LIN {X 0,Y 156.4,Z 371.31,A -85,B 0,C 180,E1 -29332.253,E2 -29332.253} C_VEL
LIN {X 0,Y 156.384,Z 371.279,A -85,B 0,C 180,E1 -29334.844,E2 -29334.844} C_VEL
LIN {X 0,Y 156.569,Z 371.648,A -85,B 0,C 180,E1 -29337.428,E2 -29337.428} C_VEL
LIN {X 0,Y 156.555,Z 373.641,A -85,B 0,C 180,E1 -29340.209,E2 -29340.209} C_VEL
LIN {X 0,Y 155.258,Z 377.324,A -85,B 0,C 180,E1 -29340.488,E2 -29340.488} C_VEL
LIN {X 0,Y 149.876,Z 389.562,A -85,B 0,C 180,E1 -29341.234,E2 -29341.234} C_VEL
LIN {X 0,Y 144.167,Z 399.757,A -85,B 0,C 180,E1 -29342.148,E2 -29342.148} C_VEL
LIN {X 0,Y 137.568,Z 409.301,A -85,B 0,C 180,E1 -29343.179,E2 -29343.179} C_VEL
LIN {X 0,Y 133.867,Z 413.861,A -85,B 0,C 180,E1 -29343.493,E2 -29343.493} C_VEL
LIN {X 0,Y 126.954,Z 420.984,A -85,B 0,C 180,E1 -29343.346,E2 -29343.346} C_VEL
LIN {X 0,Y 119.532,Z 427.573,A -85,B 0,C 180,E1 -29343.286,E2 -29343.286} C_VEL
LIN {X 0,Y 115.039,Z 431.197,A -85,B 0,C 180,E1 -29343.819,E2 -29343.819} C_VEL
LIN {X 0,Y 105.964,Z 437.725,A -85,B 0,C 180,E1 -29345.853,E2 -29345.853} C_VEL
LIN {X 0,Y 96.194,Z 443.469,A -85,B 0,C 180,E1 -29348.403,E2 -29348.403} C_VEL
LIN {X 0,Y 86.151,Z 448.159,A -85,B 0,C 180,E1 -29351.809,E2 -29351.809} C_VEL
LIN {X 0,Y 76.542,Z 451.58,A -85,B 0,C 180,E1 -29355.991,E2 -29355.991} C_VEL
LIN {X 0,Y 67.777,Z 453.839,A -85,B 0,C 180,E1 -29361.075,E2 -29361.075} C_VEL
LIN {X 0,Y 58.641,Z 455.229,A -85,B 0,C 180,E1 -29368.648,E2 -29368.648} C_VEL
LIN {X 0,Y 52.297,Z 455.5,A -85,B 0,C 180,E1 -29376.277,E2 -29376.277} C_VEL
LIN {X 0,Y 45.048,Z 454.461,A -85,B 0,C 180,E1 -29391.27,E2 -29391.27} C_VEL
LIN {X 0,Y 42.636,Z 453.317,A -85,B 0,C 180,E1 -29400.374,E2 -29400.374} C_VEL
LIN {X 0,Y 41.077,Z 450.774,A -85,B 0,C 180,E1 -29415.141,E2 -29415.141} C_VEL
LIN {X 0,Y 42.17,Z 447.189,A -85,B 0,C 180,E1 -29430.011,E2 -29430.011} C_VEL
LIN {X 0,Y 45.323,Z 442.498,A -85,B 0,C 180,E1 -29443.46,E2 -29443.46} C_VEL
LIN {X 0,Y 50.177,Z 436.573,A -85,B 0,C 180,E1 -29454.856,E2 -29454.856} C_VEL
LIN {X 0,Y 56.499,Z 429.187,A -85,B 0,C 180,E1 -29464.049,E2 -29464.049} C_VEL
LIN {X 0,Y 62.629,Z 421.633,A -85,B 0,C 180,E1 -29470.193,E2 -29470.193} C_VEL
LIN {X 0,Y 69.244,Z 412.469,A -85,B 0,C 180,E1 -29475.282,E2 -29475.282} C_VEL
LIN {X 0,Y 75.578,Z 402.269,A -85,B 0,C 180,E1 -29479.081,E2 -29479.081} C_VEL
LIN {X 0,Y 81.46,Z 390.96,A -85,B 0,C 180,E1 -29481.939,E2 -29481.939} C_VEL
LIN {X 0,Y 85.753,Z 380.375,A -85,B 0,C 180,E1 -29483.986,E2 -29483.986} C_VEL
LIN {X 0,Y 88.852,Z 370.817,A -85,B 0,C 180,E1 -29485.293,E2 -29485.293} C_VEL
LIN {X 0,Y 88.467,Z 370.007,A -85,B 0,C 180,E1 -29486.212,E2 -29486.212} C_VEL
LIN {X 0,Y 84.653,Z 375.313,A -85,B 0,C 180,E1 -29488.741,E2 -29488.741} C_VEL
LIN {X 0,Y 82.326,Z 378.124,A -85,B 0,C 180,E1 -29490.602,E2 -29490.602} C_VEL
LIN {X 0,Y 77.718,Z 385.279,A -85,B 0,C 180,E1 -29493.117,E2 -29493.117} C_VEL
LIN {X 0,Y 73.643,Z 390.721,A -85,B 0,C 180,E1 -29496.07,E2 -29496.07} C_VEL
LIN {X 0,Y 69.306,Z 395.953,A -85,B 0,C 180,E1 -29500.486,E2 -29500.486} C_VEL
LIN {X 0,Y 66.79,Z 398.707,A -85,B 0,C 180,E1 -29504.746,E2 -29504.746} C_VEL
LIN {X 0,Y 65.658,Z 400.025,A -85,B 0,C 180,E1 -29507.637,E2 -29507.637} C_VEL
LIN {X 0,Y 61.447,Z 406.178,A -85,B 0,C 180,E1 -29515.077,E2 -29515.077} C_VEL
LIN {X 0,Y 59.957,Z 408.868,A -85,B 0,C 180,E1 -29519.998,E2 -29519.998} C_VEL
LIN {X 0,Y 59.696,Z 412.054,A -85,B 0,C 180,E1 -29529.306,E2 -29529.306} C_VEL
LIN {X 0,Y 58.943,Z 418.506,A -85,B 0,C 180,E1 -29540.958,E2 -29540.958} C_VEL
LIN {X 0,Y 61.299,Z 422.846,A -85,B 0,C 180,E1 -29551.058,E2 -29551.058} C_VEL
LIN {X 0,Y 66.387,Z 425.676,A -85,B 0,C 180,E1 -29559.432,E2 -29559.432} C_VEL
LIN {X 0,Y 65.129,Z 427.629,A -85,B 0,C 180,E1 -29560.932,E2 -29560.932} C_VEL
LIN {X 0,Y 58.025,Z 434.595,A -85,B 0,C 180,E1 -29565.847,E2 -29565.847} C_VEL
LIN {X 0,Y 50.876,Z 441.526,A -85,B 0,C 180,E1 -29574.039,E2 -29574.039} C_VEL
LIN {X 0,Y 46.337,Z 446.235,A -85,B 0,C 180,E1 -29582.924,E2 -29582.924} C_VEL
LIN {X 0,Y 42.935,Z 450.806,A -85,B 0,C 180,E1 -29595.776,E2 -29595.776} C_VEL
LIN {X 0,Y 41.947,Z 454.261,A -85,B 0,C 180,E1 -29609.989,E2 -29609.989} C_VEL
LIN {X 0,Y 41.814,Z 455.932,A -85,B 0,C 180,E1 -29619.665,E2 -29619.665} C_VEL
LIN {X 0,Y 44.823,Z 458.027,A -85,B 0,C 180,E1 -29638.048,E2 -29638.048} C_VEL
LIN {X 0,Y 47.781,Z 458.503,A -85,B 0,C 180,E1 -29646.029,E2 -29646.029} C_VEL
LIN {X 0,Y 56.157,Z 458.254,A -85,B 0,C 180,E1 -29658.655,E2 -29658.655} C_VEL
LIN {X 0,Y 66.548,Z 456.484,A -85,B 0,C 180,E1 -29667.644,E2 -29667.644} C_VEL
LIN {X 0,Y 72.208,Z 454.987,A -85,B 0,C 180,E1 -29671.146,E2 -29671.146} C_VEL
LIN {X 0,Y 81.173,Z 451.969,A -85,B 0,C 180,E1 -29675.367,E2 -29675.367} C_VEL
LIN {X 0,Y 90.543,Z 447.926,A -85,B 0,C 180,E1 -29678.648,E2 -29678.648} C_VEL
LIN {X 0,Y 101.823,Z 441.734,A -85,B 0,C 180,E1 -29681.617,E2 -29681.617} C_VEL
LIN {X 0,Y 111.69,Z 435.017,A -85,B 0,C 180,E1 -29683.641,E2 -29683.641} C_VEL
LIN {X 0,Y 120.018,Z 428.188,A -85,B 0,C 180,E1 -29685.047,E2 -29685.047} C_VEL
LIN {X 0,Y 128.391,Z 419.99,A -85,B 0,C 180,E1 -29686.301,E2 -29686.301} C_VEL
LIN {X 0,Y 136.884,Z 409.9,A -85,B 0,C 180,E1 -29687.278,E2 -29687.278} C_VEL
LIN {X 0,Y 144.569,Z 398.566,A -85,B 0,C 180,E1 -29688.015,E2 -29688.015} C_VEL
LIN {X 0,Y 150.579,Z 387.394,A -85,B 0,C 180,E1 -29688.544,E2 -29688.544} C_VEL
LIN {X 0,Y 153.767,Z 379.997,A -85,B 0,C 180,E1 -29688.827,E2 -29688.827} C_VEL
LIN {X 0,Y 154.098,Z 378.981,A -85,B 0,C 180,E1 -29689.157,E2 -29689.157} C_VEL
LIN {X 0,Y 154.001,Z 378.017,A -85,B 0,C 180,E1 -29692.132,E2 -29692.132} C_VEL
LIN {X 0,Y 153.959,Z 377.955,A -85,B 0,C 180,E1 -29694.762,E2 -29694.762} C_VEL
LIN {X 0,Y 154,Z 378.711,A -85,B 0,C 180,E1 -29697.73,E2 -29697.73} C_VEL
LIN {X 0,Y 152.902,Z 381.549,A -85,B 0,C 180,E1 -29698.062,E2 -29698.062} C_VEL
LIN {X 0,Y 147.616,Z 392.5,A -85,B 0,C 180,E1 -29698.73,E2 -29698.73} C_VEL
LIN {X 0,Y 140.553,Z 404.019,A -85,B 0,C 180,E1 -29699.702,E2 -29699.702} C_VEL
LIN {X 0,Y 132.658,Z 414.293,A -85,B 0,C 180,E1 -29700.794,E2 -29700.794} C_VEL
LIN {X 0,Y 123.085,Z 424.288,A -85,B 0,C 180,E1 -29702.343,E2 -29702.343} C_VEL
LIN {X 0,Y 115.039,Z 431.197,A -85,B 0,C 180,E1 -29703.819,E2 -29703.819} C_VEL
LIN {X 0,Y 110.384,Z 434.655,A -85,B 0,C 180,E1 -29704.426,E2 -29704.426} C_VEL
LIN {X 0,Y 101.975,Z 439.939,A -85,B 0,C 180,E1 -29704.627,E2 -29704.627} C_VEL
LIN {X 0,Y 93.209,Z 444.505,A -85,B 0,C 180,E1 -29704.971,E2 -29704.971} C_VEL
LIN {X 0,Y 88.028,Z 446.834,A -85,B 0,C 180,E1 -29705.963,E2 -29705.963} C_VEL
LIN {X 0,Y 78.299,Z 450.562,A -85,B 0,C 180,E1 -29709.164,E2 -29709.164} C_VEL
LIN {X 0,Y 71.797,Z 452.509,A -85,B 0,C 180,E1 -29711.83,E2 -29711.83} C_VEL
LIN {X 0,Y 65.475,Z 454.015,A -85,B 0,C 180,E1 -29715.001,E2 -29715.001} C_VEL
LIN {X 0,Y 54.483,Z 455.57,A -85,B 0,C 180,E1 -29722.769,E2 -29722.769} C_VEL
LIN {X 0,Y 48.298,Z 455.832,A -85,B 0,C 180,E1 -29729.2,E2 -29729.2} C_VEL
LIN {X 0,Y 43.512,Z 455.567,A -85,B 0,C 180,E1 -29736.156,E2 -29736.156} C_VEL
LIN {X 0,Y 38.983,Z 454.745,A -85,B 0,C 180,E1 -29746.152,E2 -29746.152} C_VEL
LIN {X 0,Y 34.502,Z 452.265,A -85,B 0,C 180,E1 -29765.973,E2 -29765.973} C_VEL
LIN {X 0,Y 34.273,Z 449.12,A -85,B 0,C 180,E1 -29784.128,E2 -29784.128} C_VEL
LIN {X 0,Y 36.969,Z 444.898,A -85,B 0,C 180,E1 -29800.971,E2 -29800.971} C_VEL
LIN {X 0,Y 41.814,Z 439.512,A -85,B 0,C 180,E1 -29814.858,E2 -29814.858} C_VEL
LIN {X 0,Y 48.329,Z 432.775,A -85,B 0,C 180,E1 -29825.579,E2 -29825.579} C_VEL
LIN {X 0,Y 55.995,Z 424.373,A -85,B 0,C 180,E1 -29833.665,E2 -29833.665} C_VEL
LIN {X 0,Y 63,Z 415.704,A -85,B 0,C 180,E1 -29838.861,E2 -29838.861} C_VEL
LIN {X 0,Y 70.402,Z 405.048,A -85,B 0,C 180,E1 -29843.009,E2 -29843.009} C_VEL
LIN {X 0,Y 76.535,Z 394.349,A -85,B 0,C 180,E1 -29845.745,E2 -29845.745} C_VEL
LIN {X 0,Y 79.81,Z 387.444,A -85,B 0,C 180,E1 -29847.116,E2 -29847.116} C_VEL
LIN {X 0,Y 79.516,Z 387.02,A -85,B 0,C 180,E1 -29847.972,E2 -29847.972} C_VEL
LIN {X 0,Y 74.252,Z 393.462,A -85,B 0,C 180,E1 -29850.764,E2 -29850.764} C_VEL
LIN {X 0,Y 69.473,Z 398.568,A -85,B 0,C 180,E1 -29854.317,E2 -29854.317} C_VEL
LIN {X 0,Y 65.913,Z 402.042,A -85,B 0,C 180,E1 -29858.086,E2 -29858.086} C_VEL
LIN {X 0,Y 62.721,Z 404.943,A -85,B 0,C 180,E1 -29863.731,E2 -29863.731} C_VEL
LIN {X 0,Y 58.027,Z 410.485,A -85,B 0,C 180,E1 -29870.805,E2 -29870.805} C_VEL
LIN {X 0,Y 55.959,Z 413.213,A -85,B 0,C 180,E1 -29876.037,E2 -29876.037} C_VEL
LIN {X 0,Y 54.662,Z 416.981,A -85,B 0,C 180,E1 -29887.385,E2 -29887.385} C_VEL
LIN {X 0,Y 53.417,Z 422.478,A -85,B 0,C 180,E1 -29898.885,E2 -29898.885} C_VEL
LIN {X 0,Y 55.357,Z 426.811,A -85,B 0,C 180,E1 -29910.518,E2 -29910.518} C_VEL
LIN {X 0,Y 58.393,Z 428.778,A -85,B 0,C 180,E1 -29916.996,E2 -29916.996} C_VEL
LIN {X 0,Y 50.417,Z 436.169,A -85,B 0,C 180,E1 -29922.946,E2 -29922.946} C_VEL
LIN {X 0,Y 44.233,Z 441.735,A -85,B 0,C 180,E1 -29930.527,E2 -29930.527} C_VEL
LIN {X 0,Y 38.535,Z 447.18,A -85,B 0,C 180,E1 -29942.861,E2 -29942.861} C_VEL
LIN {X 0,Y 35.368,Z 451.453,A -85,B 0,C 180,E1 -29958.526,E2 -29958.526} C_VEL
LIN {X 0,Y 34.861,Z 453.696,A -85,B 0,C 180,E1 -29969.987,E2 -29969.987} C_VEL
LIN {X 0,Y 34.827,Z 455.438,A -85,B 0,C 180,E1 -29981.629,E2 -29981.629} C_VEL
LIN {X 0,Y 38.665,Z 457.615,A -85,B 0,C 180,E1 -30003.032,E2 -30003.032} C_VEL
LIN {X 0,Y 46.691,Z 458.274,A -85,B 0,C 180,E1 -30018.801,E2 -30018.801} C_VEL
LIN {X 0,Y 57.221,Z 457.338,A -85,B 0,C 180,E1 -30029.273,E2 -30029.273} C_VEL
LIN {X 0,Y 69.052,Z 454.878,A -85,B 0,C 180,E1 -30036.332,E2 -30036.332} C_VEL
LIN {X 0,Y 78.478,Z 451.931,A -85,B 0,C 180,E1 -30040.087,E2 -30040.087} C_VEL
LIN {X 0,Y 88.204,Z 447.974,A -85,B 0,C 180,E1 -30042.95,E2 -30042.95} C_VEL
LIN {X 0,Y 98.142,Z 442.893,A -85,B 0,C 180,E1 -30045.163,E2 -30045.163} C_VEL
LIN {X 0,Y 108.2,Z 436.508,A -85,B 0,C 180,E1 -30046.964,E2 -30046.964} C_VEL
LIN {X 0,Y 118.391,Z 428.578,A -85,B 0,C 180,E1 -30048.354,E2 -30048.354} C_VEL
LIN {X 0,Y 126.905,Z 420.521,A -85,B 0,C 180,E1 -30049.399,E2 -30049.399} C_VEL
LIN {X 0,Y 135.504,Z 410.688,A -85,B 0,C 180,E1 -30050.193,E2 -30050.193} C_VEL
LIN {X 0,Y 143.159,Z 399.774,A -85,B 0,C 180,E1 -30050.772,E2 -30050.772} C_VEL
LIN {X 0,Y 149.87,Z 387.705,A -85,B 0,C 180,E1 -30051.236,E2 -30051.236} C_VEL
LIN {X 0,Y 150.401,Z 386.6,A -85,B 0,C 180,E1 -30051.275,E2 -30051.275} C_VEL
LIN {X 0,Y 151.219,Z 384.614,A -85,B 0,C 180,E1 -30051.986,E2 -30051.986} C_VEL
LIN {X 0,Y 151.157,Z 384.597,A -85,B 0,C 180,E1 -30055.312,E2 -30055.312} C_VEL
LIN {X 0,Y 150.66,Z 385.733,A -85,B 0,C 180,E1 -30055.592,E2 -30055.592} C_VEL
LIN {X 0,Y 144.371,Z 397.448,A -85,B 0,C 180,E1 -30056.274,E2 -30056.274} C_VEL
LIN {X 0,Y 137.393,Z 407.735,A -85,B 0,C 180,E1 -30057.069,E2 -30057.069} C_VEL
LIN {X 0,Y 130.093,Z 416.564,A -85,B 0,C 180,E1 -30057.945,E2 -30057.945} C_VEL
LIN {X 0,Y 121.238,Z 425.413,A -85,B 0,C 180,E1 -30059.163,E2 -30059.163} C_VEL
LIN {X 0,Y 110.695,Z 433.897,A -85,B 0,C 180,E1 -30060.839,E2 -30060.839} C_VEL
LIN {X 0,Y 100.268,Z 440.649,A -85,B 0,C 180,E1 -30062.887,E2 -30062.887} C_VEL
LIN {X 0,Y 91.696,Z 445.155,A -85,B 0,C 180,E1 -30064.939,E2 -30064.939} C_VEL
LIN {X 0,Y 88.028,Z 446.834,A -85,B 0,C 180,E1 -30065.963,E2 -30065.963} C_VEL
LIN {X 0,Y 82.761,Z 448.953,A -85,B 0,C 180,E1 -30067.113,E2 -30067.113} C_VEL
LIN {X 0,Y 73.38,Z 451.955,A -85,B 0,C 180,E1 -30068.05,E2 -30068.05} C_VEL
LIN {X 0,Y 63.849,Z 454.195,A -85,B 0,C 180,E1 -30069.298,E2 -30069.298} C_VEL
LIN {X 0,Y 58.437,Z 455.085,A -85,B 0,C 180,E1 -30071.281,E2 -30071.281} C_VEL
LIN {X 0,Y 50.936,Z 455.914,A -85,B 0,C 180,E1 -30076.021,E2 -30076.021} C_VEL
LIN {X 0,Y 45.151,Z 456.14,A -85,B 0,C 180,E1 -30080.971,E2 -30080.971} C_VEL
LIN {X 0,Y 39.6,Z 455.956,A -85,B 0,C 180,E1 -30087.479,E2 -30087.479} C_VEL
LIN {X 0,Y 33.326,Z 455.026,A -85,B 0,C 180,E1 -30099.25,E2 -30099.25} C_VEL
LIN {X 0,Y 27.969,Z 452.815,A -85,B 0,C 180,E1 -30119.85,E2 -30119.85} C_VEL
LIN {X 0,Y 27.023,Z 449.758,A -85,B 0,C 180,E1 -30142.545,E2 -30142.545} C_VEL
LIN {X 0,Y 29.943,Z 445.621,A -85,B 0,C 180,E1 -30163.59,E2 -30163.59} C_VEL
LIN {X 0,Y 36.554,Z 439.323,A -85,B 0,C 180,E1 -30181.933,E2 -30181.933} C_VEL
LIN {X 0,Y 44.061,Z 432.474,A -85,B 0,C 180,E1 -30192.693,E2 -30192.693} C_VEL
LIN {X 0,Y 51.075,Z 425.472,A -85,B 0,C 180,E1 -30199.197,E2 -30199.197} C_VEL
LIN {X 0,Y 58.577,Z 416.977,A -85,B 0,C 180,E1 -30204.094,E2 -30204.094} C_VEL
LIN {X 0,Y 65.275,Z 408.121,A -85,B 0,C 180,E1 -30207.427,E2 -30207.427} C_VEL
LIN {X 0,Y 68.189,Z 403.722,A -85,B 0,C 180,E1 -30208.742,E2 -30208.742} C_VEL
LIN {X 0,Y 68.918,Z 402.36,A -85,B 0,C 180,E1 -30209.342,E2 -30209.342} C_VEL
LIN {X 0,Y 63.714,Z 406.759,A -85,B 0,C 180,E1 -30213.816,E2 -30213.816} C_VEL
LIN {X 0,Y 59.897,Z 409.646,A -85,B 0,C 180,E1 -30219.388,E2 -30219.388} C_VEL
LIN {X 0,Y 55.228,Z 414.152,A -85,B 0,C 180,E1 -30225.254,E2 -30225.254} C_VEL
LIN {X 0,Y 51.801,Z 417.679,A -85,B 0,C 180,E1 -30232.2,E2 -30232.2} C_VEL
LIN {X 0,Y 49.42,Z 421.752,A -85,B 0,C 180,E1 -30245.366,E2 -30245.366} C_VEL
LIN {X 0,Y 47.797,Z 426.491,A -85,B 0,C 180,E1 -30257.1,E2 -30257.1} C_VEL
LIN {X 0,Y 49.29,Z 430.523,A -85,B 0,C 180,E1 -30269.94,E2 -30269.94} C_VEL
LIN {X 0,Y 50.186,Z 431.333,A -85,B 0,C 180,E1 -30272.82,E2 -30272.82} C_VEL
LIN {X 0,Y 48.924,Z 432.719,A -85,B 0,C 180,E1 -30274.294,E2 -30274.294} C_VEL
LIN {X 0,Y 40.327,Z 439.869,A -85,B 0,C 180,E1 -30282.196,E2 -30282.196} C_VEL
LIN {X 0,Y 32.395,Z 446.487,A -85,B 0,C 180,E1 -30297.139,E2 -30297.139} C_VEL
LIN {X 0,Y 28.459,Z 450.847,A -85,B 0,C 180,E1 -30315.687,E2 -30315.687} C_VEL
LIN {X 0,Y 27.76,Z 453.131,A -85,B 0,C 180,E1 -30329.984,E2 -30329.984} C_VEL
LIN {X 0,Y 27.893,Z 454.917,A -85,B 0,C 180,E1 -30344.577,E2 -30344.577} C_VEL
LIN {X 0,Y 29.713,Z 456.275,A -85,B 0,C 180,E1 -30358.216,E2 -30358.216} C_VEL
LIN {X 0,Y 37.205,Z 457.757,A -85,B 0,C 180,E1 -30379.059,E2 -30379.059} C_VEL
LIN {X 0,Y 47.943,Z 457.737,A -85,B 0,C 180,E1 -30391.568,E2 -30391.568} C_VEL
LIN {X 0,Y 60.136,Z 456.121,A -85,B 0,C 180,E1 -30399.199,E2 -30399.199} C_VEL
LIN {X 0,Y 66.51,Z 454.742,A -85,B 0,C 180,E1 -30401.969,E2 -30401.969} C_VEL
LIN {X 0,Y 76.348,Z 451.871,A -85,B 0,C 180,E1 -30405.114,E2 -30405.114} C_VEL
LIN {X 0,Y 86.39,Z 447.999,A -85,B 0,C 180,E1 -30407.455,E2 -30407.455} C_VEL
LIN {X 0,Y 96.57,Z 443.016,A -85,B 0,C 180,E1 -30409.232,E2 -30409.232} C_VEL
LIN {X 0,Y 106.824,Z 436.772,A -85,B 0,C 180,E1 -30410.673,E2 -30410.673} C_VEL
LIN {X 0,Y 117.17,Z 428.969,A -85,B 0,C 180,E1 -30411.738,E2 -30411.738} C_VEL
LIN {X 0,Y 125.797,Z 421.052,A -85,B 0,C 180,E1 -30412.562,E2 -30412.562} C_VEL
LIN {X 0,Y 134.481,Z 411.397,A -85,B 0,C 180,E1 -30413.16,E2 -30413.16} C_VEL
LIN {X 0,Y 141.451,Z 401.94,A -85,B 0,C 180,E1 -30413.537,E2 -30413.537} C_VEL
LIN {X 0,Y 141.399,Z 401.999,A -85,B 0,C 180,E1 -30413.723,E2 -30413.723} C_VEL
LIN {X 0,Y 133.27,Z 412.765,A -85,B 0,C 180,E1 -30414.45,E2 -30414.45} C_VEL
LIN {X 0,Y 125.161,Z 421.52,A -85,B 0,C 180,E1 -30415.293,E2 -30415.293} C_VEL
LIN {X 0,Y 116.801,Z 429,A -85,B 0,C 180,E1 -30416.244,E2 -30416.244} C_VEL
LIN {X 0,Y 107.267,Z 436.069,A -85,B 0,C 180,E1 -30417.542,E2 -30417.542} C_VEL
LIN {X 0,Y 98.399,Z 441.468,A -85,B 0,C 180,E1 -30418.977,E2 -30418.977} C_VEL
LIN {X 0,Y 87.857,Z 446.669,A -85,B 0,C 180,E1 -30421.075,E2 -30421.075} C_VEL
LIN {X 0,Y 77.465,Z 450.611,A -85,B 0,C 180,E1 -30423.743,E2 -30423.743} C_VEL
LIN {X 0,Y 70.652,Z 452.603,A -85,B 0,C 180,E1 -30425.949,E2 -30425.949} C_VEL
LIN {X 0,Y 63.958,Z 454.161,A -85,B 0,C 180,E1 -30428.571,E2 -30428.571} C_VEL
LIN {X 0,Y 58.437,Z 455.085,A -85,B 0,C 180,E1 -30431.281,E2 -30431.281} C_VEL
LIN {X 0,Y 53.057,Z 455.8,A -85,B 0,C 180,E1 -30433.681,E2 -30433.681} C_VEL
LIN {X 0,Y 43.505,Z 456.321,A -85,B 0,C 180,E1 -30436.814,E2 -30436.814} C_VEL
LIN {X 0,Y 34.122,Z 456.06,A -85,B 0,C 180,E1 -30441.645,E2 -30441.645} C_VEL
LIN {X 0,Y 29.3,Z 455.471,A -85,B 0,C 180,E1 -30447.775,E2 -30447.775} C_VEL
LIN {X 0,Y 21.953,Z 453.335,A -85,B 0,C 180,E1 -30470.215,E2 -30470.215} C_VEL
LIN {X 0,Y 19.819,Z 450.365,A -85,B 0,C 180,E1 -30499.81,E2 -30499.81} C_VEL
LIN {X 0,Y 22.982,Z 446.33,A -85,B 0,C 180,E1 -30527.827,E2 -30527.827} C_VEL
LIN {X 0,Y 30.726,Z 440.141,A -85,B 0,C 180,E1 -30548.996,E2 -30548.996} C_VEL
LIN {X 0,Y 39.11,Z 433.403,A -85,B 0,C 180,E1 -30559.811,E2 -30559.811} C_VEL
LIN {X 0,Y 48.304,Z 424.999,A -85,B 0,C 180,E1 -30566.799,E2 -30566.799} C_VEL
LIN {X 0,Y 56.314,Z 416.328,A -85,B 0,C 180,E1 -30570.896,E2 -30570.896} C_VEL
LIN {X 0,Y 57.932,Z 414.399,A -85,B 0,C 180,E1 -30571.602,E2 -30571.602} C_VEL
LIN {X 0,Y 57.483,Z 413.986,A -85,B 0,C 180,E1 -30574.216,E2 -30574.216} C_VEL
LIN {X 0,Y 49.692,Z 420.22,A -85,B 0,C 180,E1 -30583.567,E2 -30583.567} C_VEL
LIN {X 0,Y 46.478,Z 423.056,A -85,B 0,C 180,E1 -30591.301,E2 -30591.301} C_VEL
LIN {X 0,Y 44.594,Z 425.344,A -85,B 0,C 180,E1 -30599.998,E2 -30599.998} C_VEL
LIN {X 0,Y 42.692,Z 428.404,A -85,B 0,C 180,E1 -30608.925,E2 -30608.925} C_VEL
LIN {X 0,Y 42.279,Z 432.649,A -85,B 0,C 180,E1 -30623.891,E2 -30623.891} C_VEL
LIN {X 0,Y 42.309,Z 434.236,A -85,B 0,C 180,E1 -30628.689,E2 -30628.689} C_VEL
LIN {X 0,Y 33.12,Z 441.153,A -85,B 0,C 180,E1 -30637.252,E2 -30637.252} C_VEL
LIN {X 0,Y 24.671,Z 447.382,A -85,B 0,C 180,E1 -30655.247,E2 -30655.247} C_VEL
LIN {X 0,Y 20.939,Z 451.46,A -85,B 0,C 180,E1 -30680.317,E2 -30680.317} C_VEL
LIN {X 0,Y 20.67,Z 452.566,A -85,B 0,C 180,E1 -30689.979,E2 -30689.979} C_VEL
LIN {X 0,Y 23.668,Z 455.811,A -85,B 0,C 180,E1 -30726.409,E2 -30726.409} C_VEL
LIN {X 0,Y 32.976,Z 457.385,A -85,B 0,C 180,E1 -30748.459,E2 -30748.459} C_VEL
LIN {X 0,Y 44.987,Z 457.46,A -85,B 0,C 180,E1 -30759.581,E2 -30759.581} C_VEL
LIN {X 0,Y 57.989,Z 455.94,A -85,B 0,C 180,E1 -30765.793,E2 -30765.793} C_VEL
LIN {X 0,Y 71.432,Z 452.869,A -85,B 0,C 180,E1 -30769.658,E2 -30769.658} C_VEL
LIN {X 0,Y 81.691,Z 449.425,A -85,B 0,C 180,E1 -30771.594,E2 -30771.594} C_VEL
LIN {X 0,Y 92.038,Z 444.918,A -85,B 0,C 180,E1 -30773.022,E2 -30773.022} C_VEL
LIN {X 0,Y 98.966,Z 441.231,A -85,B 0,C 180,E1 -30773.784,E2 -30773.784} C_VEL
LIN {X 0,Y 98.808,Z 441.269,A -85,B 0,C 180,E1 -30774.69,E2 -30774.69} C_VEL
LIN {X 0,Y 88.032,Z 446.59,A -85,B 0,C 180,E1 -30776.235,E2 -30776.235} C_VEL
LIN {X 0,Y 77.335,Z 450.649,A -85,B 0,C 180,E1 -30778.275,E2 -30778.275} C_VEL
LIN {X 0,Y 70.006,Z 452.765,A -85,B 0,C 180,E1 -30780.001,E2 -30780.001} C_VEL
LIN {X 0,Y 63.28,Z 454.298,A -85,B 0,C 180,E1 -30781.941,E2 -30781.941} C_VEL
LIN {X 0,Y 55.426,Z 455.568,A -85,B 0,C 180,E1 -30784.849,E2 -30784.849} C_VEL
LIN {X 0,Y 43.058,Z 456.446,A -85,B 0,C 180,E1 -30791.725,E2 -30791.725} C_VEL
LIN {X 0,Y 36.778,Z 456.324,A -85,B 0,C 180,E1 -30797.208,E2 -30797.208} C_VEL
LIN {X 0,Y 29.3,Z 455.471,A -85,B 0,C 180,E1 -30807.775,E2 -30807.775} C_VEL
LIN {X 0,Y 24.931,Z 454.646,A -85,B 0,C 180,E1 -30816.003,E2 -30816.003} C_VEL
LIN {X 0,Y 17.694,Z 452.738,A -85,B 0,C 180,E1 -30833.818,E2 -30833.818} C_VEL
LIN {X 0,Y 13.915,Z 450.653,A -85,B 0,C 180,E1 -30858.595,E2 -30858.595} C_VEL
LIN {X 0,Y 14.134,Z 448.71,A -85,B 0,C 180,E1 -30881.727,E2 -30881.727} C_VEL
LIN {X 0,Y 14.908,Z 447.981,A -85,B 0,C 180,E1 -30888.351,E2 -30888.351} C_VEL
LIN {X 0,Y 21.224,Z 443.765,A -85,B 0,C 180,E1 -30911.502,E2 -30911.502} C_VEL
LIN {X 0,Y 30.145,Z 437.831,A -85,B 0,C 180,E1 -30924.71,E2 -30924.71} C_VEL
LIN {X 0,Y 39.817,Z 430.438,A -85,B 0,C 180,E1 -30931.973,E2 -30931.973} C_VEL
LIN {X 0,Y 46.477,Z 424.502,A -85,B 0,C 180,E1 -30935.156,E2 -30935.156} C_VEL
LIN {X 0,Y 44.779,Z 425.207,A -85,B 0,C 180,E1 -30940.368,E2 -30940.368} C_VEL
LIN {X 0,Y 40.916,Z 428.001,A -85,B 0,C 180,E1 -30950.107,E2 -30950.107} C_VEL
LIN {X 0,Y 39.73,Z 429.108,A -85,B 0,C 180,E1 -30954.923,E2 -30954.923} C_VEL
LIN {X 0,Y 35.997,Z 434.875,A -85,B 0,C 180,E1 -30977.021,E2 -30977.021} C_VEL
LIN {X 0,Y 35.539,Z 436.132,A -85,B 0,C 180,E1 -30981.573,E2 -30981.573} C_VEL
LIN {X 0,Y 27.834,Z 441.356,A -85,B 0,C 180,E1 -30987.872,E2 -30987.872} C_VEL
LIN {X 0,Y 19.279,Z 446.689,A -85,B 0,C 180,E1 -31003.158,E2 -31003.158} C_VEL
LIN {X 0,Y 14.013,Z 450.855,A -85,B 0,C 180,E1 -31035.444,E2 -31035.444} C_VEL
LIN {X 0,Y 13.582,Z 452.001,A -85,B 0,C 180,E1 -31049.967,E2 -31049.967} C_VEL
LIN {X 0,Y 14.589,Z 453.866,A -85,B 0,C 180,E1 -31078.764,E2 -31078.764} C_VEL
LIN {X 0,Y 23.79,Z 456.381,A -85,B 0,C 180,E1 -31112.365,E2 -31112.365} C_VEL
LIN {X 0,Y 36.358,Z 457.275,A -85,B 0,C 180,E1 -31125.079,E2 -31125.079} C_VEL
LIN {X 0,Y 49.812,Z 456.674,A -85,B 0,C 180,E1 -31130.919,E2 -31130.919} C_VEL
LIN {X 0,Y 63.564,Z 454.459,A -85,B 0,C 180,E1 -31134.243,E2 -31134.243} C_VEL
LIN {X 0,Y 63.463,Z 454.436,A -85,B 0,C 180,E1 -31135.242,E2 -31135.242} C_VEL
LIN {X 0,Y 56.298,Z 455.657,A -85,B 0,C 180,E1 -31136.902,E2 -31136.902} C_VEL
LIN {X 0,Y 46.52,Z 456.594,A -85,B 0,C 180,E1 -31140.002,E2 -31140.002} C_VEL
LIN {X 0,Y 35.303,Z 456.673,A -85,B 0,C 180,E1 -31145.64,E2 -31145.64} C_VEL
LIN {X 0,Y 24.404,Z 455.583,A -85,B 0,C 180,E1 -31156.742,E2 -31156.742} C_VEL
LIN {X 0,Y 16.979,Z 453.846,A -85,B 0,C 180,E1 -31174.169,E2 -31174.169} C_VEL
LIN {X 0,Y 12.718,Z 450.958,A -85,B 0,C 180,E1 -31213.997,E2 -31213.997} C_VEL
LIN {X 0,Y 14.908,Z 447.981,A -85,B 0,C 180,E1 -31248.351,E2 -31248.351} C_VEL
LIN {X 0,Y 17.704,Z 445.729,A -85,B 0,C 180,E1 -31264.806,E2 -31264.806} C_VEL
LIN {X 0,Y 23.042,Z 441.578,A -85,B 0,C 180,E1 -31285.455,E2 -31285.455} C_VEL
LIN {X 0,Y 29.793,Z 436.745,A -85,B 0,C 180,E1 -31297.668,E2 -31297.668} C_VEL
LIN {X 0,Y 34.436,Z 433.4,A -85,B 0,C 180,E1 -31300.841,E2 -31300.841} C_VEL
LIN {X 0,Y 37.008,Z 431.425,A -85,B 0,C 180,E1 -31301.757,E2 -31301.757} C_VEL
LIN {X 0,Y 36.695,Z 431.57,A -85,B 0,C 180,E1 -31303.304,E2 -31303.304} C_VEL
LIN {X 0,Y 33.471,Z 433.884,A -85,B 0,C 180,E1 -31313.971,E2 -31313.971} C_VEL
LIN {X 0,Y 30.728,Z 436.548,A -85,B 0,C 180,E1 -31325.546,E2 -31325.546} C_VEL
LIN {X 0,Y 28.74,Z 438.458,A -85,B 0,C 180,E1 -31331.931,E2 -31331.931} C_VEL
LIN {X 0,Y 18.584,Z 444.324,A -85,B 0,C 180,E1 -31338.938,E2 -31338.938} C_VEL
LIN {X 0,Y 9.489,Z 448.963,A -85,B 0,C 180,E1 -31362.147,E2 -31362.147} C_VEL
LIN {X 0,Y 6.493,Z 451.435,A -85,B 0,C 180,E1 -31409.932,E2 -31409.932} C_VEL
LIN {X 0,Y 14.85,Z 454.838,A -85,B 0,C 180,E1 -31481.089,E2 -31481.089} C_VEL
LIN {X 0,Y 21.438,Z 455.946,A -85,B 0,C 180,E1 -31489.459,E2 -31489.459} C_VEL
LIN {X 0,Y 28.263,Z 456.639,A -85,B 0,C 180,E1 -31493.922,E2 -31493.922} C_VEL
LIN {X 0,Y 28.162,Z 456.577,A -85,B 0,C 180,E1 -31496.336,E2 -31496.336} C_VEL
LIN {X 0,Y 21.078,Z 455.68,A -85,B 0,C 180,E1 -31500.831,E2 -31500.831} C_VEL
LIN {X 0,Y 14.221,Z 454.356,A -85,B 0,C 180,E1 -31508.95,E2 -31508.95} C_VEL
LIN {X 0,Y 6.048,Z 451.553,A -85,B 0,C 180,E1 -31554.567,E2 -31554.567} C_VEL
LIN {X 0,Y 10.209,Z 447.693,A -85,B 0,C 180,E1 -31633.565,E2 -31633.565} C_VEL
LIN {X 0,Y 19.88,Z 442.712,A -85,B 0,C 180,E1 -31652.151,E2 -31652.151} C_VEL
LIN {X 0,Y 30.092,Z 436.471,A -85,B 0,C 180,E1 -31659.138,E2 -31659.138} C_VEL
LIN {X 0,Y 34.436,Z 433.4,A -85,B 0,C 180,E1 -31660.841,E2 -31660.841} C_VEL
LIN {X 0,Y 33.861,Z 433.727,A -85,B 0,C 180,E1 -31662.543,E2 -31662.543} C_VEL
LIN {X 0,Y 29.169,Z 436.8,A -85,B 0,C 180,E1 -31666.343,E2 -31666.343} C_VEL
LIN {X 0,Y 23.471,Z 440.292,A -85,B 0,C 180,E1 -31669.995,E2 -31669.995} C_VEL
LIN {X 0,Y 18.436,Z 443.101,A -85,B 0,C 180,E1 -31672.813,E2 -31672.813} C_VEL
LIN {X 0,Y 16.705,Z 443.973,A -85,B 0,C 180,E1 -31673.333,E2 -31673.333} C_VEL
LIN {X 0,Y 14.144,Z 445.251,A -85,B 0,C 180,E1 -31673.896,E2 -31673.896} C_VEL
LIN {X 0,Y 14.095,Z 445.306,A -85,B 0,C 180,E1 -31676.167,E2 -31676.167} C_VEL
LIN {X 0,Y 21.12,Z 441.754,A -85,B 0,C 180,E1 -31677.014,E2 -31677.014} C_VEL
LIN {X 0,Y 21.26,Z 441.58,A -85,B 0,C 180,E1 -31672.791,E2 -31672.791} C_VEL
LIN {X 0,Y 16.705,Z 443.973,A -85,B 0,C 180,E1 -31673.333,E2 -31673.333} C_VEL
LIN {X 0,Y 15.599,Z 445.763,A -85,B 0,C 180,E1 -31673.554,E2 -31673.554} C_VEL
LIN {X 0,Y 15.599,Z 600,A -85,B 0,C 180,E1 -31673.554,E2 -31673.554} C_VEL
LIN {X 0,Y 15.599,Z 600,A -85,B 0,C 180,E1 -31673.554,E2 -31673.554}

QRS_NEXT_CUT()

QRS_NEXT()
QRS_HOME()

END
